// TIA Portal V18 export
TYPE "UDT_OP10_Recipe_type"
   STRUCT
      Header : Struct   // Information about recipe
         RecipeName : String[50];   // name of product
         RecipeID : USInt;   // number of product for sig exch. and other processes
         "Version" : UInt;   // version of update that structure
         LastModified : DTL;   // time of last modifiacation
         PartType : String[28];   // second name for product - additional one
         PartTypeRecordNr : Int;   // PartType Record number same like recipi id for future sig exchanges etc
      END_STRUCT;
      Process : Struct   // Important process parameters how should machine act
         Timers : Struct   // Definition of times for processess
            Delay_glue_init_start : Time := T#2S;
            Delay_Medium : Time;
            Delay_Long : Time;
            Cylinder_ActTime : Time;
         END_STRUCT;
         Limits : Struct   // limitations of the values
            RetryLimit : Int;
         END_STRUCT;
         Press : Struct   // parameters for the kistler press devices
            B1_Program : Int;
            B2_Program : Int;
            Curve { S7_SetPoint := 'True'} : "UDT_Recipe_PressCurve";
         END_STRUCT;
         Vision : Struct   // camera system programs numbers
            CGlueShaftIV3_Progs : Array[1..4] of Word;
            CGlueMagnetIV3_Prog : Word;
            CGlueProgram : Int;
         END_STRUCT;
      END_STRUCT;
      "Tooling Code" : Struct   // QR CODES OF THE TOOLING FOR THE RECIPE
         A1_Table : Array[1..8] of String[128];
         A2_Table : Array[1..8] of String[128];   // ... other fixture codes Descriptive Gripper Fixture Codes
         ROB1_Shaft_Handling_Robot : Struct   // R1
            Gripper { S7_SetPoint := 'True'} : "UDT_Gripper_Fixture_Codes";
         END_STRUCT;
         ROB2_Main_Assembly_Robot : Struct   // R2
            Gripper { S7_SetPoint := 'True'} : "UDT_Gripper_Fixture_Codes";
         END_STRUCT;
         ROB3_Unloading_Robot : Struct   // R3
            Gripper { S7_SetPoint := 'True'} : "UDT_Gripper_Fixture_Codes";
         END_STRUCT;
         A1_Fixtures : Struct
            A1RingUnloadingFixtureCode : String[128];
            E1LoadingNGFixtureCode : String[128];
            ShaftScanFixtureCode : String[128];
            B1PressFixtureCode : String[128];
            CGlueFixtureCode : String[128];
            B1PressCylFixtureCode : String[128];
         END_STRUCT;
         A2_Fixtures : Struct
            A2RingUnloadingFixtureCode : String[128];
            E2UnloadingNGFixtureCode : String[128];
            B2PressFixtureCode : String[128];
            CGlueNGFixtureCode : String[128];
            B2PressCylFixtureCode : String[128];
         END_STRUCT;
      END_STRUCT;
      Motion : Struct   // ALL SERVO DRIVES PARAMETERS
         Gluing_Nozzle_Z { S7_SetPoint := 'True'} : "UDT_IAI_Axis_Positions";   // Physical Axis: IAI_A1
         Gluing_Nozzle_X { S7_SetPoint := 'True'} : "UDT_IAI_Axis_Positions";   // Physical Axis: IAI_A2
         Gluing_Nozzle_Y { S7_SetPoint := 'True'} : "UDT_IAI_Axis_Positions";   // Physical Axis: IAI_A3 CORRECTED V90 Axis Functions (from user)
         Ring_Turntable_Axis_1 { S7_SetPoint := 'True'} : "UDT_V90_Axis_Positions";   // Physical Axis: V90_A1
         Shaft_Scan_Turntable_Axis { S7_SetPoint := 'True'} : "UDT_V90_Axis_Positions";   // Physical Axis: V90_A2
         Gluing_Rotary_Jig_Axis { S7_SetPoint := 'True'} : "UDT_V90_Axis_Positions";   // Physical Axis: V90_A3
         Ring_Turntable_Axis_2 { S7_SetPoint := 'True'} : "UDT_V90_Axis_Positions";   // Physical Axis: V90_A4
      END_STRUCT;
   END_STRUCT;
END_TYPE
